{attribute 'GeneratedUsingTerminal: EL3403-0000-0017'}
{attribute addProperty BoxType "EL3403-0000-0017"}
{attribute addProperty Id "IndexAT %Q*USINT1"}
{attribute addProperty CRC "3858488880"}
{attribute addProperty Size "1"}
TYPE PM_Outputs_Channel_E5FBDE30 :
STRUCT
	{attribute addProperty Name "Index"}
	Index AT %Q* : USINT;
END_STRUCT
END_TYPE

(* stored: Version 1.2.0.0, ProductVersion 3.1.4024.9
   DUT PM_Outputs_Channel_E5FBDE30: Id {5c60313c-7b10-45a9-8f75-d3cbd103db5f} *)
